// TwinCAT 3 PLC project UdpMulticastDevice2
// libraries:
//   Tc2_Standard, * (Beckhoff Automation GmbH)
//   Tc2_System, * (Beckhoff Automation GmbH)
//   Tc2_TcpIp, * (Beckhoff Automation GmbH)
//   Tc2_Utilities, * (Beckhoff Automation GmbH)
//   Tc3_Module, * (Beckhoff Automation GmbH)
// project tree:
//   / PlcTask2.TcTTO
//   POUs/ MAIN.TcPOU, RecivedData.TcDUT
// real-time tasks:
//   TASK PlcTask2: cycle T#200000us, priority 21, ADS port 351

CONFIGURATION UdpMulticastDevice2
    RESOURCE PLC ON TwinCAT3
        TASK PlcTask2(INTERVAL := T#200000us, PRIORITY := 21);
        PROGRAM MAIN WITH PlcTask2 : MAIN;
    END_RESOURCE
END_CONFIGURATION

// ---- POUs/RecivedData.TcDUT
TYPE RecivedData :
UNION
	tbytes					:ARRAY[0..255]OF BYTE;
	tString					:STRING[255];
	tUDINT					:UDINT;
	tINT					:INT;
END_UNION
END_TYPE

// ---- POUs/MAIN.TcPOU
PROGRAM MAIN
VAR
	bEnable					: BOOL 	:= TRUE;
	nLocalPort				: UDINT := 1001;
	sLocalHost				: T_IPv4Addr := '172.16.17.48';(* Adapt local IP address to your device *)
	nRemotePort				: UDINT := 1002;
	sMulticastAddr			: T_IPv4Addr := '224.1.1.255';
	
	fbUdpCreate 			: FB_SocketUdpCreate;
	fbSocketAddMulticast 	: FB_SocketUdpAddMulticastAddress;
	fbSocketDropMulticast 	: FB_SocketUdpDropMulticastAddress;
	fbSocketSend  			: FB_SocketUdpSendTo;
	fbSocketReceive 		: FB_SocketUdpReceiveFrom;
	fbSocketClose			: FB_SocketClose;
	fbCloseAll				: FB_SocketCloseAll;
	bInitialize				: BOOL := TRUE;
	bUdpCreated				: BOOL;
	bMulticastAdded			: BOOL; 
	
	InData					:RecivedData;
	LastRecived				:RecivedData;
	NullData				:RecivedData;
	//nCounterIn 				: UDINT;
	nCounterOut 			: UDINT;
	sCounterOutAsString		: STRING;
	nState 					: INT;
END_VAR

(* On PLC reset or program download close all opened/created sockets *)
fbCloseAll( bExecute:= bInitialize );
IF fbCloseAll.bBusy OR fbCloseAll.bError THEN
	RETURN;
END_IF
bInitialize := FALSE;


CASE nState OF
0:
	IF bEnable THEN
		bUdpCreated := FALSE;
		bMulticastAdded := FALSE;
		nState := 1;
	END_IF
1:
	fbUdpCreate( bExecute := FALSE );
	fbUdpCreate( nLocalPort := nLocalPort, sLocalHost := sLocalHost, bExecute := TRUE);
	nState := 2;
2:
	fbUdpCreate( bExecute := FALSE );
	IF NOT fbUdpCreate.bBusy THEN
		IF NOT fbUdpCreate.bError THEN
			bUdpCreated := TRUE;
			fbSocketAddMulticast( bExecute := FALSE );
			fbSocketAddMulticast( hSocket := fbUdpCreate.hSocket, sMulticastAddr := sMulticastAddr, bExecute := TRUE );
			nState := 3;
		ELSE
			nState := 100;
		END_IF
	END_IF
3:
	fbSocketAddMulticast( bExecute := FALSE );
	IF NOT fbSocketAddMulticast.bBusy THEN
		IF NOT fbSocketAddMulticast.bError THEN
			bMulticastAdded := TRUE;
			nState := 4;
		ELSE
			nState := 100;
		END_IF
	END_IF
	
4:
	IF bEnable THEN
		nCounterOut := nCounterOut + 1;
		sCounterOutAsString:=TO_STRING(nCounterOut);
		fbSocketSend( bExecute := FALSE );
		fbSocketSend( nRemotePort := nRemotePort, sRemoteHost := sMulticastAddr, hSocket := fbUdpCreate.hSocket, cbLen:= SIZEOF(sCounterOutAsString), pSrc := ADR(sCounterOutAsString), bExecute := TRUE );
		nState := 5;
	ELSE
		nState := 10;
	END_IF
5:
	fbSocketSend( bExecute := FALSE );
	IF NOT fbSocketSend.bBusy THEN
		IF NOT fbSocketSend.bError THEN
			fbSocketReceive( bExecute := FALSE );
			MEMSET(destAddr:=ADR(InData) , fillByte:=0 , n:=SIZEOF(InData));
			fbSocketReceive( hSocket := fbUdpCreate.hSocket, cbLen := SIZEOF(InData), pDest := ADR(InData), bExecute := TRUE );
			nState := 6;
		ELSE
 			nState := 100;
		END_IF
	END_IF
6:	
	fbSocketReceive( bExecute := FALSE );
	IF NOT fbSocketReceive.bBusy THEN
		IF NOT fbSocketReceive.bError THEN
			IF MEMCMP(pBuf1:=ADR(InData), pBuf2:=ADR(NullData) , n:=SIZEOF(RecivedData)) <>0 THEN
				LastRecived:=InData;
			END_IF
			nState:= 4;
		ELSE
			nState := 100;
		END_IF
	END_IF

10:
	fbSocketDropMulticast( bExecute := FALSE );
	fbSocketDropMulticast( hSocket := fbUdpCreate.hSocket, sMulticastAddr := sMulticastAddr, bExecute := TRUE );
	nState := 11;
11:	
	fbSocketDropMulticast( bExecute := FALSE );
	IF NOT fbSocketDropMulticast.bBusy THEN
		bMulticastAdded := FALSE;
		IF NOT fbSocketDropMulticast.bError THEN
			nState := 20;
		ELSE
			nState := 100;
		END_IF
	END_IF

20:	
	fbSocketClose( bExecute := FALSE );
	fbSocketClose( hSocket := fbUdpCreate.hSocket, bExecute := TRUE );
	nState := 21;
21:	
	fbSocketClose( bExecute := FALSE );
	IF NOT fbSocketClose.bBusy THEN
		bUdpCreated := FALSE;
		IF NOT fbSocketClose.bError THEN
			nState := 0;	
		ELSE
			nState := 100;	
		END_IF
	END_IF
	
100:
	IF bMulticastAdded THEN
		nState := 10;
	ELSIF bUdpCreated THEN
		nState := 20;
	ELSE
		nState := 0;
	END_IF
	
END_CASE

END_PROGRAM
